{attribute addProperty BoxType "EL3681-0000-0018"}
{attribute addProperty Id "SettingsAT %I*Settings_7AA6B313162"}
{attribute addProperty CRC "3751299124"}
{attribute addProperty SizeInBites "16"}
{attribute addProperty SizeInBytes "2"}
TYPE SAI_Range_DF984834 :
STRUCT
	{attribute addProperty Name "Settings"}
	Settings AT %I* : Settings_7AA6B313;
END_STRUCT
END_TYPE

(* stored: Version 1.2.0.0, ProductVersion 3.1.4024.9
   DUT SAI_Range_DF984834: Id {d266938c-ad3b-4284-bb0a-3f6eb8a439e3} *)
